TYPE TasterEventType : (TASTEVT_NoOne := 0,
		TASTEVT_PositiveEdge,
		TASTEVT_NegativeEdge,
		TASTEVT_LongClick,
		TASTEVT_DoubleClick,
		TASTEVT_PositiveNegativeEdge,
		TASTEVT_End_LongClick,
		TASTEVT_TimeElapsedAfterNegativeEdge);
END_TYPE

(* stored: Version 1.1.0.1, ProductVersion 3.1.4022.7
   DUT TasterEventType: Id {94e4eb96-cb61-4c9d-9f10-a4a1f438e3f2} *)
